{attribute 'qualified_only'}
{attribute 'strict'}
{attribute 'to_string'}
TYPE E_AlarmSeverity :
(
	NoneAlarm := 0,
	InfoAlarm,
	WarningAlarm,
	ErrorAlarm
) BYTE := NoneAlarm;
END_TYPE

(* stored: Version 1.1.0.1, ProductVersion 3.1.4024.15
   DUT E_AlarmSeverity: Id {b2ecf0aa-0b63-44c2-baf1-61f189e67d83} *)
